{attribute 'GeneratedUsingTerminal: EK1100-0000-0018'}
{attribute addProperty BoxType "EK1100-0000-0018"}
{attribute addProperty Id "Beckhoff_ATH2xxxEK1122Beckhoff_ATH2xxxEK1122_61A38CAE870A_0013_ATH2000_5250_0022ATH2000_D874080E14"}
{attribute addProperty CRC "289678688"}
{attribute addProperty Size "884"}
TYPE Beckhoff_ATH2xxx_11442560 EXTENDS EK1100_1FC0878B :
STRUCT
	{attribute addProperty Name "Beckhoff ATH2xxxEK1122"}
	{attribute addProperty PreviousPort "Beckhoff ATH2xxx : B"}
	Beckhoff_ATH2xxxEK1122 : Beckhoff_ATH2xxxEK1122_61A38CAE;
	{attribute addProperty Name "A_0013(ATH2000-5250-0022)"}
	{attribute addProperty PreviousPort "Beckhoff ATH2xxxEK1122 : C"}
	A_0013_ATH2000_5250_0022 : ATH2000_D874080E;
END_STRUCT
END_TYPE

(* stored: Version 1.2.0.0, ProductVersion 3.1.4024.9
   DUT Beckhoff_ATH2xxx_11442560: Id {cb4f7768-07bb-4462-818c-690b6ea8a104} *)
